// TIA Portal V21 export
FUNCTION "GestStazione_ProntoRicevere" : Void   // FC413, LAD
{ S7_Optimized_Access := 'TRUE' }
// stored: SetENOAutomatically false
   VAR_INPUT
      AttivaChiamata : Bool;
      K_Stazione : Int;
   END_VAR
   VAR_TEMP
      ProntaChiamareNoFeedback : Bool;   // La stazione è pronta a chiamare ma manca il feedback
      StazioneRiferimentoAdditiva : Int;
      StazioneRiferimentoAdditivoPresente : Bool;
      StazioneSorgenteAdditivoPresente : Bool;
      DestinazioneAttuale : Int;
      AlmenoUnaDestInChiamata : Bool;
      ChiamataOrBypass : Bool;
      AlmenoUnaDestAttiva : Bool;
      PercorsoNonAttivato : Bool;
      PercorsoSelezionato : Bool;
      K_StazioneDestinazione : Int;
      StazioneRiferimento1_InvioAdditivo : Int;
      StazioneRiferimento2_InvioAdditivo : Int;
      BypassControlloRiferimenti : Bool;
   END_VAR
BEGIN

REGION Network 1 (SCL): Gestione della chiamata della stazione
   REGION Pulizia memorie
       #K_StazioneDestinazione :=
       #StazioneRiferimento1_InvioAdditivo :=
       #StazioneRiferimento2_InvioAdditivo :=
       #StazioneRiferimentoAdditiva := 0;

       #AlmenoUnaDestInChiamata :=
       #StazioneSorgenteAdditivoPresente :=
       #StazioneRiferimentoAdditivoPresente :=
       #PercorsoNonAttivato :=
       #PercorsoSelezionato :=
       #AlmenoUnaDestAttiva := False;
   END_REGION ;

   FOR #DestinazioneAttuale := 0 TO "K_NumStazione" DO //Sfoglio tutte le stazioni
       //Se la stazione controllata è in chiamata oppure se è bypassata (non deve aspettare la chimata di valle per chiamare)
       #ChiamataOrBypass := "Percorso".Stazione[#DestinazioneAttuale].OUT.Chiamata OR "Percorso".Stazione[#K_Stazione].Prm.ByPassChiamataDestinazione;

       IF "Percorso".Stazione[#K_Stazione].Destinazione[#DestinazioneAttuale].IN.Selezionato THEN
           #PercorsoSelezionato := True;
           IF NOT "Percorso".Stazione[#K_Stazione].Destinazione[#DestinazioneAttuale].IN.Attivo THEN
               #PercorsoNonAttivato := True;
           END_IF;
       END_IF;
       IF "Percorso".Stazione[#K_Stazione].Destinazione[#DestinazioneAttuale].IN.Attivo THEN //Se la strada verso la destinazione è attiva (quindi selezionata e caricata in lavoro)
           #AlmenoUnaDestAttiva := True;
           "Percorso".Stazione[#DestinazioneAttuale].Dati.SorgAttivaPresente := True;
           IF #ChiamataOrBypass THEN                                                                                                       //verifico che sia anche in chiamata
               #AlmenoUnaDestInChiamata := True;  //e setto la chiamata.
           END_IF;                                                                                                                         //Anche se non chiama posso salvare la K.
           #K_StazioneDestinazione := #DestinazioneAttuale;                                           //Salvo nella stazione la K che identifica la mia destinazione attiva.
           IF "Percorso".Stazione[#K_Stazione].Dati.InvioAdditivo.Abilitazione THEN                                                        //Se ho abilitato il funzionamento additivo per questa stazione
               FOR #StazioneRiferimentoAdditiva := 0 TO "K_NumStazione" DO                                                                 //Inizio a cercare la stazione partner, sfogliando tutte le stazioni
                   IF "Percorso".Stazione[#StazioneRiferimentoAdditiva].Dati.K_StazioneDestinazione = #DestinazioneAttuale THEN            //verifico che abbia la mia stessa destinazione,
                       IF #StazioneRiferimentoAdditiva <> #K_Stazione THEN                                                                 //mi assicuro di saltare la stazione attuale.
                           #StazioneSorgenteAdditivoPresente := #StazioneRiferimentoAdditivoPresente := True;                              //A questo punto posso dire di avere una stazione ed una destinazione attiva.
                           "Percorso".Stazione[#StazioneRiferimentoAdditiva].Dati.RicezioneAdditivo.K_StazioneRiferimento := #K_Stazione;  //Scrivo nella stazione che ho trovato la sorgente additivo.
                           IF #StazioneRiferimento1_InvioAdditivo = 0 THEN                                                                 //Scrivo nella stazione attuale la k della destinazione di riferimento trovata.
                               #StazioneRiferimento1_InvioAdditivo := #StazioneRiferimentoAdditiva;
                           ELSE
                               #StazioneRiferimento2_InvioAdditivo := #StazioneRiferimentoAdditiva;
                           END_IF;
                       END_IF;
                   END_IF;
               END_FOR;
           END_IF;
       END_IF;
       IF "Percorso".Stazione[#K_Stazione].Destinazione[#DestinazioneAttuale].IN.Possibile THEN    //Se questo percorso è possibile significa che
           "Percorso".Stazione[#DestinazioneAttuale].Dati.AlmenoUnaSorgenteProgettata := True;     //questa destinazione ha almeno una sorgente progettata
           "Percorso".Stazione[#K_Stazione].Dati.AlmenoUnaDestinazioneProgettata := True;          //e di conseguenza questa stazione ha almeno una destinazione progettata.
       END_IF;
   END_FOR;

   REGION Gestione timeout stazione
       "T_ON"(I_CicloCPU := "CicloScansioneCPU_I".O_rCicloCpu,
              I_StartConteggio := "Percorso".Stazione[#K_Stazione].OUT.Chiamata AND NOT "Percorso".Stazione[#K_Stazione].IN.Feedback_Run,
              IO_DatiTimer := "Percorso".Stazione[#K_Stazione].Prm.FeedbackRun.Attesa);
   END_REGION ;

   //Appoggio di seguito le tempo
   "Percorso".Stazione[#K_Stazione].Dati.InvioAdditivo.K_StazioneRiferimento1 := #StazioneRiferimento1_InvioAdditivo;
   "Percorso".Stazione[#K_Stazione].Dati.InvioAdditivo.K_StazioneRiferimento2 := #StazioneRiferimento2_InvioAdditivo;

   "Percorso".Stazione[#K_Stazione].Dati.InvioAdditivo.Attiva := #StazioneRiferimentoAdditivoPresente;
   "Percorso".Stazione["Percorso".Stazione[#K_Stazione].Dati.InvioAdditivo.K_StazioneRiferimento1].Dati.RicezioneAdditivo.Attiva :=
   "Percorso".Stazione["Percorso".Stazione[#K_Stazione].Dati.InvioAdditivo.K_StazioneRiferimento2].Dati.RicezioneAdditivo.Attiva := #StazioneSorgenteAdditivoPresente;
   "Percorso".Stazione[#K_Stazione].Dati.DestAttivaPresente := #AlmenoUnaDestAttiva;
   "Percorso".Stazione[#K_Stazione].Dati.K_StazioneDestinazione := #K_StazioneDestinazione;
END_REGION

REGION Network 2: La stazione è pronta a chiamare
   // AlmenoUnaDestInChiamata = Significa che è presente una destinazione e che mi sta chiamando oppure ho attivo il parametro che mi permette di non aspettare la chiamata della destinazione.
   // 
   // AttivaChiamata = Questo parametro viene passato da fuori com ingresso del blocco, se le condizioni sono valide, la stazione chiama.
   // 
   // Struct.Hmi.Abilita = ON/OFF presente su matrice che permette / abilita la chiamata.
   // 
   // ProntaAChiamare = La stazione è pronta a chiamare per quanto la riguarda.
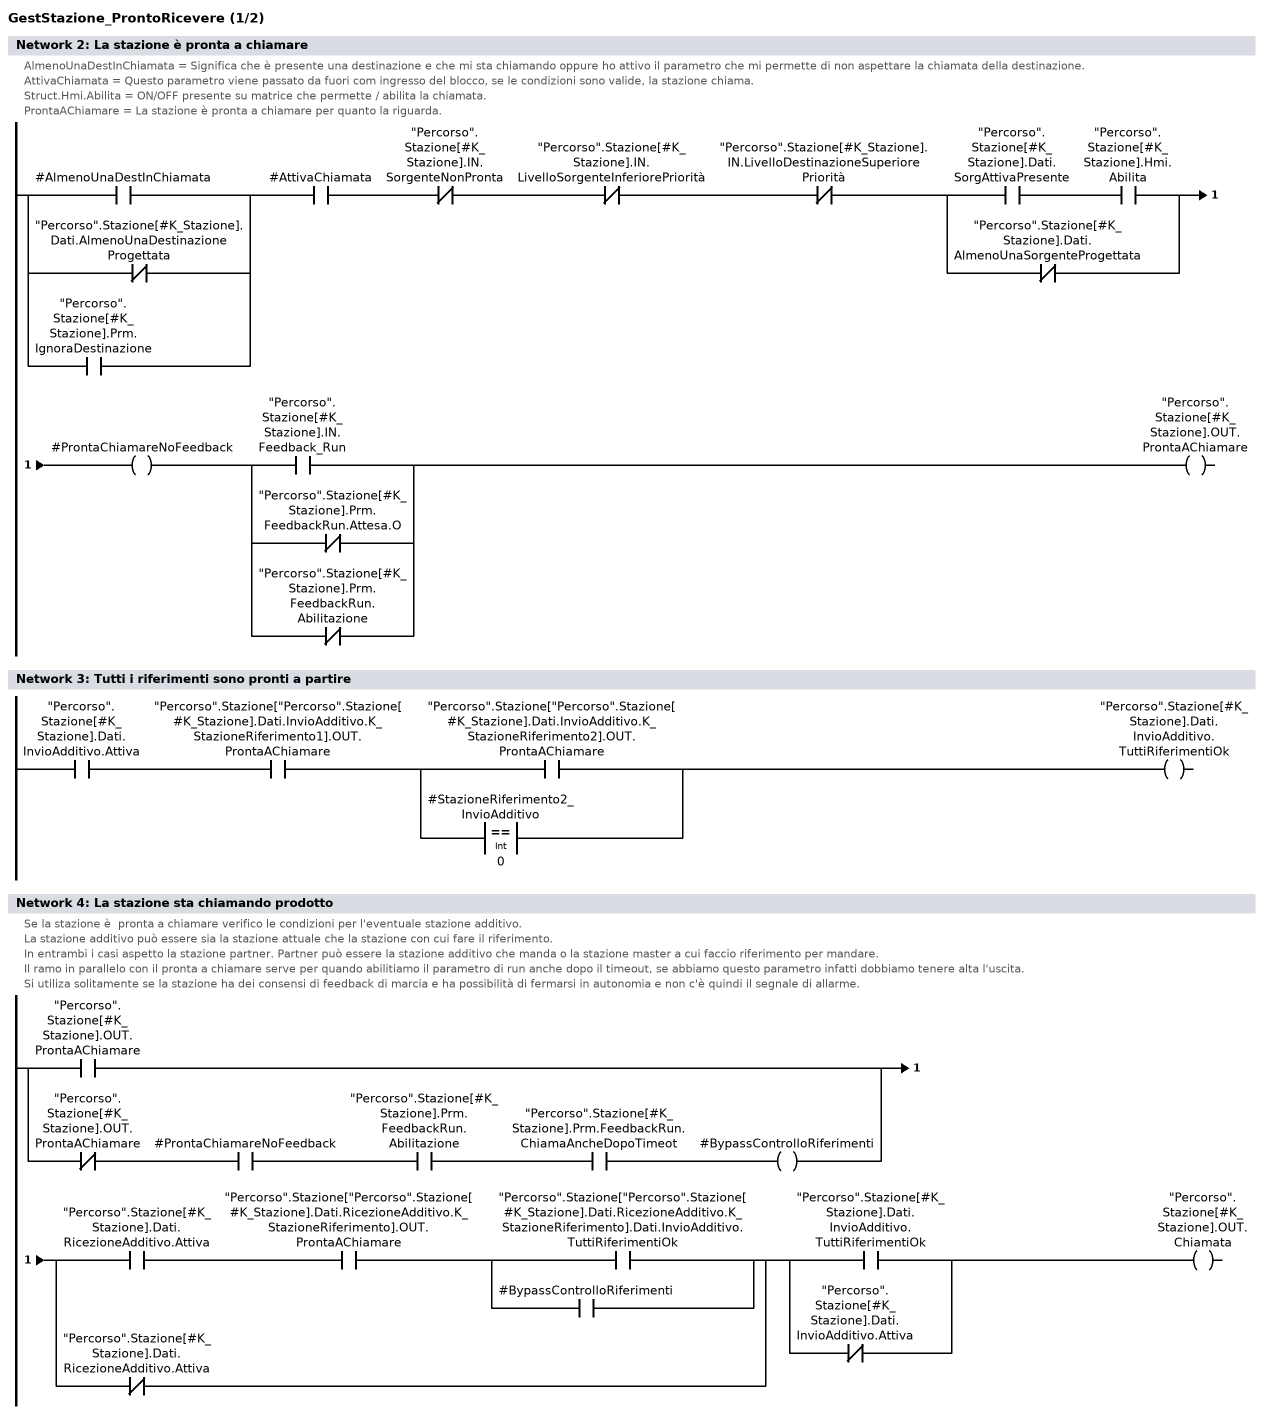
   RUNG wire#powerrail
      Contact( #AlmenoUnaDestInChiamata )
      wire#w1
      Contact( #AttivaChiamata )
      I_Contact( "Percorso".Stazione[#K_Stazione].IN.SorgenteNonPronta )
      I_Contact( "Percorso".Stazione[#K_Stazione].IN.LivelloSorgenteInferiorePriorità )
      I_Contact( "Percorso".Stazione[#K_Stazione].IN.LivelloDestinazioneSuperiorePriorità )
      wire#w2
      Contact( "Percorso".Stazione[#K_Stazione].Dati.SorgAttivaPresente )
      Contact( "Percorso".Stazione[#K_Stazione].Hmi.Abilita )
      wire#w3
      Coil( #ProntaChiamareNoFeedback )
      wire#w4
      Contact( "Percorso".Stazione[#K_Stazione].IN.Feedback_Run )
      wire#w5
      Coil( "Percorso".Stazione[#K_Stazione].OUT.ProntaAChiamare )
   END_RUNG
   RUNG wire#powerrail
      I_Contact( "Percorso".Stazione[#K_Stazione].Dati.AlmenoUnaDestinazioneProgettata )
   END_RUNG wire#w1
   RUNG wire#powerrail
      Contact( "Percorso".Stazione[#K_Stazione].Prm.IgnoraDestinazione )
   END_RUNG wire#w1
   RUNG wire#w2
      I_Contact( "Percorso".Stazione[#K_Stazione].Dati.AlmenoUnaSorgenteProgettata )
   END_RUNG wire#w3
   RUNG wire#w4
      I_Contact( "Percorso".Stazione[#K_Stazione].Prm.FeedbackRun.Attesa.O )
   END_RUNG wire#w5
   RUNG wire#w4
      I_Contact( "Percorso".Stazione[#K_Stazione].Prm.FeedbackRun.Abilitazione )
   END_RUNG wire#w5
   // the same network as SCL:
   #ProntaChiamareNoFeedback := (#AlmenoUnaDestInChiamata OR NOT "Percorso".Stazione[#K_Stazione].Dati.AlmenoUnaDestinazioneProgettata OR "Percorso".Stazione[#K_Stazione].Prm.IgnoraDestinazione) AND #AttivaChiamata AND NOT "Percorso".Stazione[#K_Stazione].IN.SorgenteNonPronta AND NOT "Percorso".Stazione[#K_Stazione].IN.LivelloSorgenteInferiorePriorità AND NOT "Percorso".Stazione[#K_Stazione].IN.LivelloDestinazioneSuperiorePriorità AND (("Percorso".Stazione[#K_Stazione].Dati.SorgAttivaPresente AND "Percorso".Stazione[#K_Stazione].Hmi.Abilita) OR NOT "Percorso".Stazione[#K_Stazione].Dati.AlmenoUnaSorgenteProgettata);
   "Percorso".Stazione[#K_Stazione].OUT.ProntaAChiamare := #ProntaChiamareNoFeedback AND ("Percorso".Stazione[#K_Stazione].IN.Feedback_Run OR NOT "Percorso".Stazione[#K_Stazione].Prm.FeedbackRun.Attesa.O OR NOT "Percorso".Stazione[#K_Stazione].Prm.FeedbackRun.Abilitazione);
END_REGION

REGION Network 3: Tutti i riferimenti sono pronti a partire
   RUNG wire#powerrail
      Contact( "Percorso".Stazione[#K_Stazione].Dati.InvioAdditivo.Attiva )
      Contact( "Percorso".Stazione["Percorso".Stazione[#K_Stazione].Dati.InvioAdditivo.K_StazioneRiferimento1].OUT.ProntaAChiamare )
      wire#w1
      Contact( "Percorso".Stazione["Percorso".Stazione[#K_Stazione].Dati.InvioAdditivo.K_StazioneRiferimento2].OUT.ProntaAChiamare )
      wire#w2
      Coil( "Percorso".Stazione[#K_Stazione].Dati.InvioAdditivo.TuttiRiferimentiOk )
   END_RUNG
   RUNG wire#w1
      { S7_Templates := "SrcType := Int" } EQ_Contact(in1 := #StazioneRiferimento2_InvioAdditivo, in2 := 0)
   END_RUNG wire#w2
   // the same network as SCL:
   "Percorso".Stazione[#K_Stazione].Dati.InvioAdditivo.TuttiRiferimentiOk := "Percorso".Stazione[#K_Stazione].Dati.InvioAdditivo.Attiva AND "Percorso".Stazione["Percorso".Stazione[#K_Stazione].Dati.InvioAdditivo.K_StazioneRiferimento1].OUT.ProntaAChiamare AND ("Percorso".Stazione["Percorso".Stazione[#K_Stazione].Dati.InvioAdditivo.K_StazioneRiferimento2].OUT.ProntaAChiamare OR (#StazioneRiferimento2_InvioAdditivo = 0));
END_REGION

REGION Network 4: La stazione sta chiamando prodotto
   // Se la stazione è  pronta a chiamare verifico le condizioni per l'eventuale stazione additivo.
   // La stazione additivo può essere sia la stazione attuale che la stazione con cui fare il riferimento.
   // In entrambi i casi aspetto la stazione partner. Partner può essere la stazione additivo che manda o la stazione master a cui faccio riferimento per mandare.
   // 
   // Il ramo in parallelo con il pronta a chiamare serve per quando abilitiamo il parametro di run anche dopo il timeout, se abbiamo questo parametro infatti dobbiamo tenere alta l'uscita.
   // Si utiliza solitamente se la stazione ha dei consensi di feedback di marcia e ha possibilità di fermarsi in autonomia e non c'è quindi il segnale di allarme.
   RUNG wire#powerrail
      Contact( "Percorso".Stazione[#K_Stazione].OUT.ProntaAChiamare )
      wire#w1
      Contact( "Percorso".Stazione[#K_Stazione].Dati.RicezioneAdditivo.Attiva )
      Contact( "Percorso".Stazione["Percorso".Stazione[#K_Stazione].Dati.RicezioneAdditivo.K_StazioneRiferimento].OUT.ProntaAChiamare )
      wire#w2
      Contact( "Percorso".Stazione["Percorso".Stazione[#K_Stazione].Dati.RicezioneAdditivo.K_StazioneRiferimento].Dati.InvioAdditivo.TuttiRiferimentiOk )
      wire#w3
      Contact( "Percorso".Stazione[#K_Stazione].Dati.InvioAdditivo.TuttiRiferimentiOk )
      wire#w4
      Coil( "Percorso".Stazione[#K_Stazione].OUT.Chiamata )
   END_RUNG
   RUNG wire#powerrail
      I_Contact( "Percorso".Stazione[#K_Stazione].OUT.ProntaAChiamare )
      Contact( #ProntaChiamareNoFeedback )
      Contact( "Percorso".Stazione[#K_Stazione].Prm.FeedbackRun.Abilitazione )
      Contact( "Percorso".Stazione[#K_Stazione].Prm.FeedbackRun.ChiamaAncheDopoTimeot )
      Coil( #BypassControlloRiferimenti )
   END_RUNG wire#w1
   RUNG wire#w2
      Contact( #BypassControlloRiferimenti )
   END_RUNG wire#w3
   RUNG wire#w1
      I_Contact( "Percorso".Stazione[#K_Stazione].Dati.RicezioneAdditivo.Attiva )
   END_RUNG wire#w3
   RUNG wire#w3
      I_Contact( "Percorso".Stazione[#K_Stazione].Dati.InvioAdditivo.Attiva )
   END_RUNG wire#w4
   // the same network as SCL:
   #BypassControlloRiferimenti := NOT "Percorso".Stazione[#K_Stazione].OUT.ProntaAChiamare AND #ProntaChiamareNoFeedback AND "Percorso".Stazione[#K_Stazione].Prm.FeedbackRun.Abilitazione AND "Percorso".Stazione[#K_Stazione].Prm.FeedbackRun.ChiamaAncheDopoTimeot;
   "Percorso".Stazione[#K_Stazione].OUT.Chiamata := ("Percorso".Stazione[#K_Stazione].OUT.ProntaAChiamare OR #BypassControlloRiferimenti) AND (("Percorso".Stazione[#K_Stazione].Dati.RicezioneAdditivo.Attiva AND "Percorso".Stazione["Percorso".Stazione[#K_Stazione].Dati.RicezioneAdditivo.K_StazioneRiferimento].OUT.ProntaAChiamare AND ("Percorso".Stazione["Percorso".Stazione[#K_Stazione].Dati.RicezioneAdditivo.K_StazioneRiferimento].Dati.InvioAdditivo.TuttiRiferimentiOk OR #BypassControlloRiferimenti)) OR NOT "Percorso".Stazione[#K_Stazione].Dati.RicezioneAdditivo.Attiva) AND ("Percorso".Stazione[#K_Stazione].Dati.InvioAdditivo.TuttiRiferimentiOk OR NOT "Percorso".Stazione[#K_Stazione].Dati.InvioAdditivo.Attiva);
END_REGION

REGION Network 5: Diagnostica
   // Se la stazione è  pronta a chiamare verifico le condizioni per l'eventuale stazione additivo.
   // La stazione additivo può essere sia la stazione attuale che la stazione con cui fare il riferimento.
   // In entrambi i casi aspetto la stazione partner. Partner può essere la stazione additivo che manda o la stazione master a cui faccio riferimento per mandare.
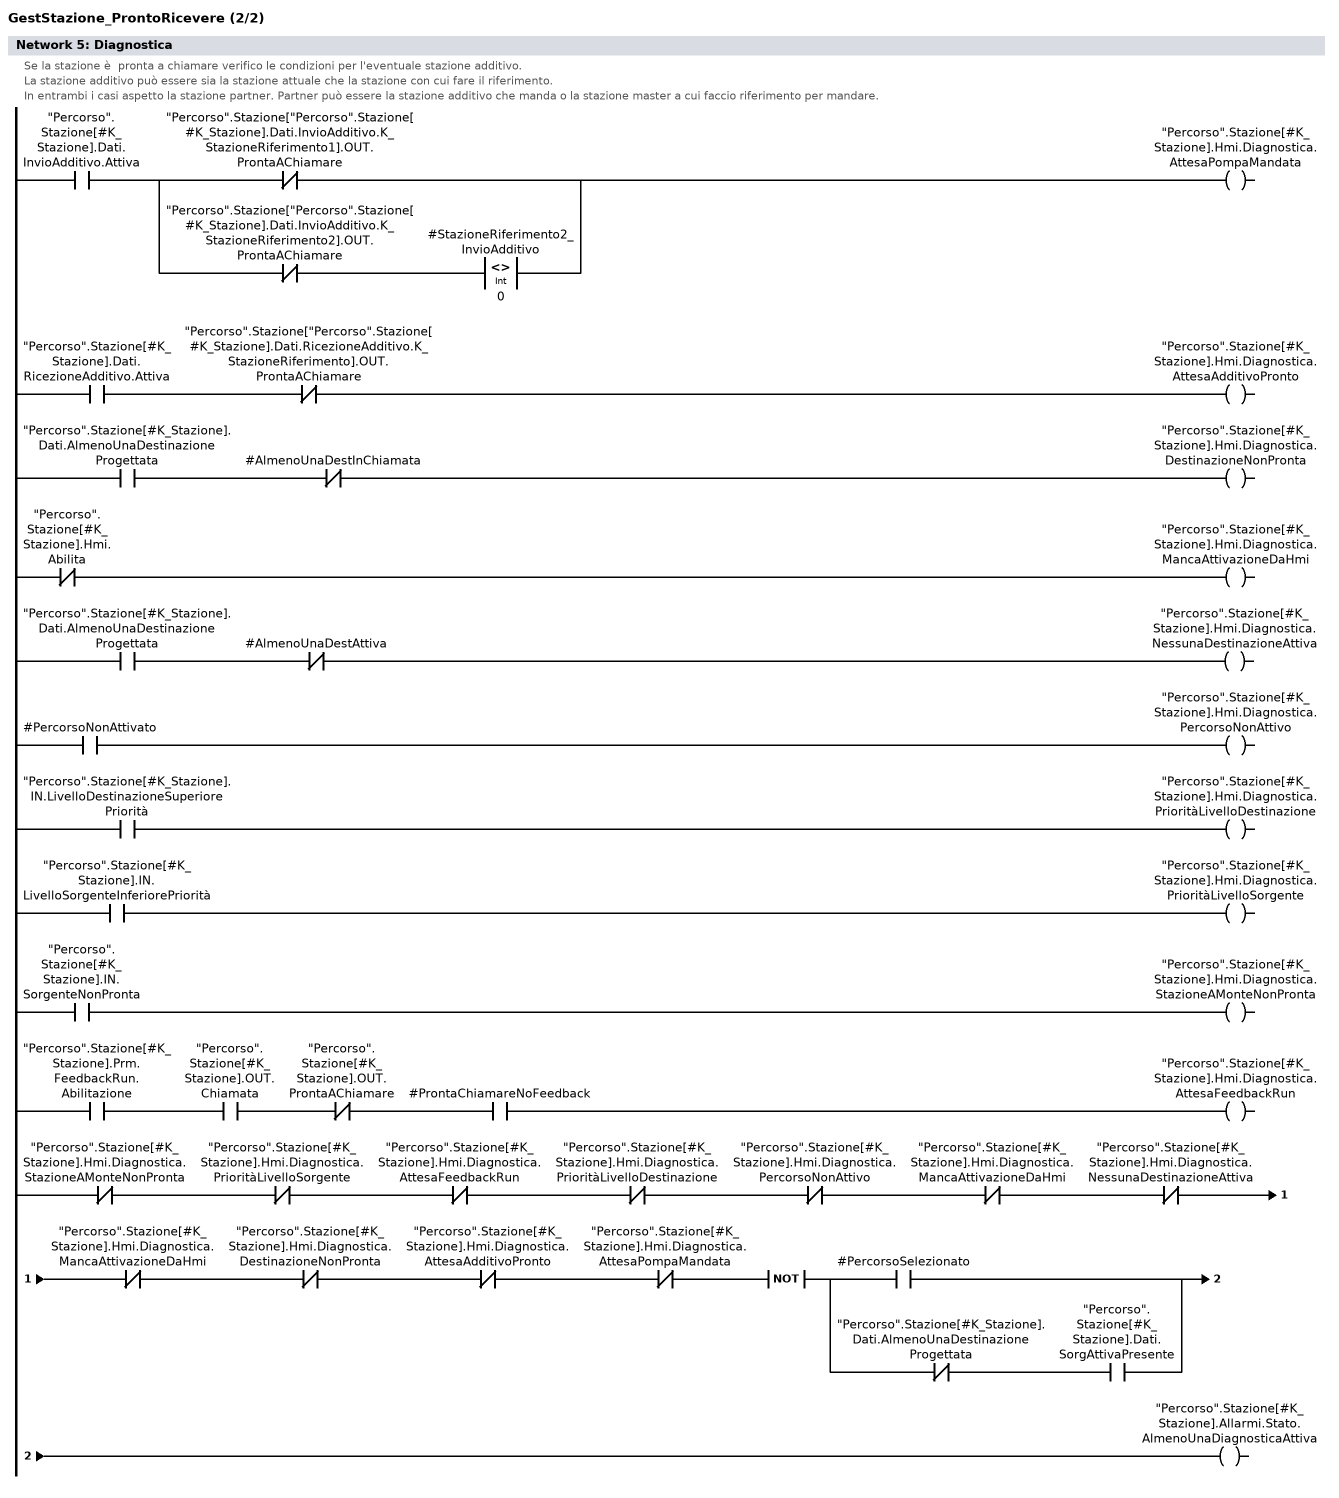
   RUNG wire#powerrail
      Contact( "Percorso".Stazione[#K_Stazione].Dati.InvioAdditivo.Attiva )
      wire#w1
      I_Contact( "Percorso".Stazione["Percorso".Stazione[#K_Stazione].Dati.InvioAdditivo.K_StazioneRiferimento1].OUT.ProntaAChiamare )
      wire#w2
      Coil( "Percorso".Stazione[#K_Stazione].Hmi.Diagnostica.AttesaPompaMandata )
   END_RUNG
   RUNG wire#w1
      I_Contact( "Percorso".Stazione["Percorso".Stazione[#K_Stazione].Dati.InvioAdditivo.K_StazioneRiferimento2].OUT.ProntaAChiamare )
      { S7_Templates := "SrcType := Int" } NE_Contact(in1 := #StazioneRiferimento2_InvioAdditivo, in2 := 0)
   END_RUNG wire#w2
   RUNG wire#powerrail
      Contact( "Percorso".Stazione[#K_Stazione].Dati.RicezioneAdditivo.Attiva )
      I_Contact( "Percorso".Stazione["Percorso".Stazione[#K_Stazione].Dati.RicezioneAdditivo.K_StazioneRiferimento].OUT.ProntaAChiamare )
      Coil( "Percorso".Stazione[#K_Stazione].Hmi.Diagnostica.AttesaAdditivoPronto )
   END_RUNG
   RUNG wire#powerrail
      Contact( "Percorso".Stazione[#K_Stazione].Dati.AlmenoUnaDestinazioneProgettata )
      I_Contact( #AlmenoUnaDestInChiamata )
      Coil( "Percorso".Stazione[#K_Stazione].Hmi.Diagnostica.DestinazioneNonPronta )
   END_RUNG
   RUNG wire#powerrail
      I_Contact( "Percorso".Stazione[#K_Stazione].Hmi.Abilita )
      Coil( "Percorso".Stazione[#K_Stazione].Hmi.Diagnostica.MancaAttivazioneDaHmi )
   END_RUNG
   RUNG wire#powerrail
      Contact( "Percorso".Stazione[#K_Stazione].Dati.AlmenoUnaDestinazioneProgettata )
      I_Contact( #AlmenoUnaDestAttiva )
      Coil( "Percorso".Stazione[#K_Stazione].Hmi.Diagnostica.NessunaDestinazioneAttiva )
   END_RUNG
   RUNG wire#powerrail
      Contact( #PercorsoNonAttivato )
      Coil( "Percorso".Stazione[#K_Stazione].Hmi.Diagnostica.PercorsoNonAttivo )
   END_RUNG
   RUNG wire#powerrail
      Contact( "Percorso".Stazione[#K_Stazione].IN.LivelloDestinazioneSuperiorePriorità )
      Coil( "Percorso".Stazione[#K_Stazione].Hmi.Diagnostica.PrioritàLivelloDestinazione )
   END_RUNG
   RUNG wire#powerrail
      Contact( "Percorso".Stazione[#K_Stazione].IN.LivelloSorgenteInferiorePriorità )
      Coil( "Percorso".Stazione[#K_Stazione].Hmi.Diagnostica.PrioritàLivelloSorgente )
   END_RUNG
   RUNG wire#powerrail
      Contact( "Percorso".Stazione[#K_Stazione].IN.SorgenteNonPronta )
      Coil( "Percorso".Stazione[#K_Stazione].Hmi.Diagnostica.StazioneAMonteNonPronta )
   END_RUNG
   RUNG wire#powerrail
      Contact( "Percorso".Stazione[#K_Stazione].Prm.FeedbackRun.Abilitazione )
      Contact( "Percorso".Stazione[#K_Stazione].OUT.Chiamata )
      I_Contact( "Percorso".Stazione[#K_Stazione].OUT.ProntaAChiamare )
      Contact( #ProntaChiamareNoFeedback )
      Coil( "Percorso".Stazione[#K_Stazione].Hmi.Diagnostica.AttesaFeedbackRun )
   END_RUNG
   RUNG wire#powerrail
      I_Contact( "Percorso".Stazione[#K_Stazione].Hmi.Diagnostica.StazioneAMonteNonPronta )
      I_Contact( "Percorso".Stazione[#K_Stazione].Hmi.Diagnostica.PrioritàLivelloSorgente )
      I_Contact( "Percorso".Stazione[#K_Stazione].Hmi.Diagnostica.AttesaFeedbackRun )
      I_Contact( "Percorso".Stazione[#K_Stazione].Hmi.Diagnostica.PrioritàLivelloDestinazione )
      I_Contact( "Percorso".Stazione[#K_Stazione].Hmi.Diagnostica.PercorsoNonAttivo )
      I_Contact( "Percorso".Stazione[#K_Stazione].Hmi.Diagnostica.MancaAttivazioneDaHmi )
      I_Contact( "Percorso".Stazione[#K_Stazione].Hmi.Diagnostica.NessunaDestinazioneAttiva )
      I_Contact( "Percorso".Stazione[#K_Stazione].Hmi.Diagnostica.MancaAttivazioneDaHmi )
      I_Contact( "Percorso".Stazione[#K_Stazione].Hmi.Diagnostica.DestinazioneNonPronta )
      I_Contact( "Percorso".Stazione[#K_Stazione].Hmi.Diagnostica.AttesaAdditivoPronto )
      I_Contact( "Percorso".Stazione[#K_Stazione].Hmi.Diagnostica.AttesaPompaMandata )
      Not()
      wire#w3
      Contact( #PercorsoSelezionato )
      wire#w4
      Coil( "Percorso".Stazione[#K_Stazione].Allarmi.Stato.AlmenoUnaDiagnosticaAttiva )
   END_RUNG
   RUNG wire#w3
      I_Contact( "Percorso".Stazione[#K_Stazione].Dati.AlmenoUnaDestinazioneProgettata )
      Contact( "Percorso".Stazione[#K_Stazione].Dati.SorgAttivaPresente )
   END_RUNG wire#w4
   // the same network as SCL:
   "Percorso".Stazione[#K_Stazione].Hmi.Diagnostica.AttesaPompaMandata := "Percorso".Stazione[#K_Stazione].Dati.InvioAdditivo.Attiva AND (NOT "Percorso".Stazione["Percorso".Stazione[#K_Stazione].Dati.InvioAdditivo.K_StazioneRiferimento1].OUT.ProntaAChiamare OR (NOT "Percorso".Stazione["Percorso".Stazione[#K_Stazione].Dati.InvioAdditivo.K_StazioneRiferimento2].OUT.ProntaAChiamare AND (#StazioneRiferimento2_InvioAdditivo <> 0)));
   "Percorso".Stazione[#K_Stazione].Hmi.Diagnostica.AttesaAdditivoPronto := "Percorso".Stazione[#K_Stazione].Dati.RicezioneAdditivo.Attiva AND NOT "Percorso".Stazione["Percorso".Stazione[#K_Stazione].Dati.RicezioneAdditivo.K_StazioneRiferimento].OUT.ProntaAChiamare;
   "Percorso".Stazione[#K_Stazione].Hmi.Diagnostica.DestinazioneNonPronta := "Percorso".Stazione[#K_Stazione].Dati.AlmenoUnaDestinazioneProgettata AND NOT #AlmenoUnaDestInChiamata;
   "Percorso".Stazione[#K_Stazione].Hmi.Diagnostica.MancaAttivazioneDaHmi := NOT "Percorso".Stazione[#K_Stazione].Hmi.Abilita;
   "Percorso".Stazione[#K_Stazione].Hmi.Diagnostica.NessunaDestinazioneAttiva := "Percorso".Stazione[#K_Stazione].Dati.AlmenoUnaDestinazioneProgettata AND NOT #AlmenoUnaDestAttiva;
   "Percorso".Stazione[#K_Stazione].Hmi.Diagnostica.PercorsoNonAttivo := #PercorsoNonAttivato;
   "Percorso".Stazione[#K_Stazione].Hmi.Diagnostica.PrioritàLivelloDestinazione := "Percorso".Stazione[#K_Stazione].IN.LivelloDestinazioneSuperiorePriorità;
   "Percorso".Stazione[#K_Stazione].Hmi.Diagnostica.PrioritàLivelloSorgente := "Percorso".Stazione[#K_Stazione].IN.LivelloSorgenteInferiorePriorità;
   "Percorso".Stazione[#K_Stazione].Hmi.Diagnostica.StazioneAMonteNonPronta := "Percorso".Stazione[#K_Stazione].IN.SorgenteNonPronta;
   "Percorso".Stazione[#K_Stazione].Hmi.Diagnostica.AttesaFeedbackRun := "Percorso".Stazione[#K_Stazione].Prm.FeedbackRun.Abilitazione AND "Percorso".Stazione[#K_Stazione].OUT.Chiamata AND NOT "Percorso".Stazione[#K_Stazione].OUT.ProntaAChiamare AND #ProntaChiamareNoFeedback;
   "Percorso".Stazione[#K_Stazione].Allarmi.Stato.AlmenoUnaDiagnosticaAttiva := NOT (NOT "Percorso".Stazione[#K_Stazione].Hmi.Diagnostica.StazioneAMonteNonPronta AND NOT "Percorso".Stazione[#K_Stazione].Hmi.Diagnostica.PrioritàLivelloSorgente AND NOT "Percorso".Stazione[#K_Stazione].Hmi.Diagnostica.AttesaFeedbackRun AND NOT "Percorso".Stazione[#K_Stazione].Hmi.Diagnostica.PrioritàLivelloDestinazione AND NOT "Percorso".Stazione[#K_Stazione].Hmi.Diagnostica.PercorsoNonAttivo AND NOT "Percorso".Stazione[#K_Stazione].Hmi.Diagnostica.MancaAttivazioneDaHmi AND NOT "Percorso".Stazione[#K_Stazione].Hmi.Diagnostica.NessunaDestinazioneAttiva AND NOT "Percorso".Stazione[#K_Stazione].Hmi.Diagnostica.MancaAttivazioneDaHmi AND NOT "Percorso".Stazione[#K_Stazione].Hmi.Diagnostica.DestinazioneNonPronta AND NOT "Percorso".Stazione[#K_Stazione].Hmi.Diagnostica.AttesaAdditivoPronto AND NOT "Percorso".Stazione[#K_Stazione].Hmi.Diagnostica.AttesaPompaMandata) AND (#PercorsoSelezionato OR (NOT "Percorso".Stazione[#K_Stazione].Dati.AlmenoUnaDestinazioneProgettata AND "Percorso".Stazione[#K_Stazione].Dati.SorgAttivaPresente));
END_REGION

REGION Network 6 (SCL): Pulisco la memoria dopo averla letta
   //Ripulisco le memorie di arresto chiamata a causa delle priorità
   IF NOT "Percorso".Stazione[#K_Stazione].Dati.GestionePrioritàAttiva.DaDestinazione THEN
       "Percorso".Stazione[#K_Stazione].IN.LivelloDestinazioneSuperiorePriorità := False;
   END_IF;
   IF NOT "Percorso".Stazione[#K_Stazione].Dati.GestionePrioritàAttiva.DaSorgente THEN
       "Percorso".Stazione[#K_Stazione].IN.LivelloSorgenteInferiorePriorità := False;
   END_IF;
   "Percorso".Stazione[#K_Stazione].Dati.LivelloTank_PerMotore := "Percorso".Stazione[#K_Stazione].Dati.LivelloTank_DaSorgente;
   "Percorso".Stazione[#K_Stazione].Dati.IntMinLivelloTank_PerMotore := "Percorso".Stazione[#K_Stazione].Dati.IntMinLivelloTank_DaSorgente;
   //Ripulisco le memorie dopo averle lette
   "Percorso".Stazione[#K_Stazione].IN.SorgenteNonPronta :=
   "Percorso".Stazione[#K_Stazione].Dati.SorgAttivaPresente :=
   "Percorso".Stazione[#K_Stazione].Dati.RicezioneAdditivo.Attiva :=
   "Percorso".Stazione[#K_Stazione].Dati.GestionePrioritàAttiva.DaDestinazione :=
   "Percorso".Stazione[#K_Stazione].Dati.GestionePrioritàAttiva.DaSorgente :=
   "Percorso".Stazione[#K_Stazione].Dati.IntMinLivelloTank_DaSorgente := False;
   "Percorso".Stazione[#K_Stazione].Dati.LivelloTank_DaSorgente := 0;
END_REGION

REGION Network 7 (SCL): Riferimenti incrociati
   // "Percorso".Stazione[#K_Stazione].Rif_Inc.K_Analogica := #K_Analogica;
   // "Percorso".Stazione[#K_Stazione].Rif_Inc.K_Paratia := #K_Paratia;
   // "Percorso".Stazione[#K_Stazione].Rif_Inc.K_Motore := #K_Motore;
   // "Percorso".Stazione[#K_Stazione].Rif_Inc.K_Pompa := #K_Pompa;
END_REGION
END_FUNCTION
